{attribute 'linkalways'} 
{attribute 'no_explicit_call' := 'This FB is a CLASS and must be accessed using methods or properties'}
{attribute 'enable_dynamic_creation'}
FUNCTION_BLOCK _DINT EXTENDS NumericDatatypeBase
VAR
	localData : DINT;
	activeData : REFERENCE TO DINT REF= localData;
END_VAR

PROPERTY PUBLIC Address : PVOID
GET
Address := ADR(activeData);
END_GET
END_PROPERTY

METHOD PUBLIC ClearReference
VAR_INPUT
END_VAR
activeData REF= localData;
END_METHOD

METHOD PUBLIC Clone : I_Datatype
VAR
    pClone : POINTER TO _DINT;
END_VAR
pClone := __NEW(_DINT(InitialValue := Value));
Clone := pClone^;
END_METHOD

METHOD FB_init : BOOL
VAR_INPUT
	bInitRetains : BOOL; // if TRUE, the retain variables are initialized (warm start / cold start)
	bInCopyCode : BOOL;  // if TRUE, the instance afterwards gets moved into the copy code (online change)
	InitialValue : DINT;
END_VAR
localData := InitialValue;
END_METHOD

PROPERTY PUBLIC IsFloat : BOOL
GET
IsFloat := FALSE;
END_GET
END_PROPERTY

PROPERTY PUBLIC IsSigned : BOOL
GET
IsSigned := TRUE;
END_GET
END_PROPERTY

METHOD PUBLIC MakeReferenceTo
VAR_INPUT
	ReferenceTarget : REFERENCE TO DINT;
END_VAR
activeData REF= ReferenceTarget;
END_METHOD

PROPERTY PUBLIC MaxValue : DINT
GET
MaxValue := DatatypeLimits.DINT_MAX_VALUE;
END_GET
END_PROPERTY

PROPERTY PUBLIC MinValue : DINT
GET
MinValue := DatatypeLimits.DINT_MIN_VALUE;
END_GET
END_PROPERTY

METHOD PROTECTED SerializeMaxValue
VAR_INPUT
	Serializer : I_Serializer;
END_VAR
Serializer.AddDint(MaxValue);
END_METHOD

METHOD PROTECTED SerializeMinValue
VAR_INPUT
	Serializer : I_Serializer;
END_VAR
Serializer.AddDint(MinValue);
END_METHOD

METHOD PUBLIC SerializeWith
VAR_INPUT
	Serializer : I_Serializer;
END_VAR
Serializer.AddDint(activeData);
END_METHOD

PROPERTY PUBLIC Size : UDINT
GET
Size := SIZEOF(activeData);
END_GET
END_PROPERTY

METHOD TryDeserializeFrom : BOOL
VAR_INPUT
	Deserializer : I_Deserializer;
	Feedback : I_DeserializerFeedback;
END_VAR
TryDeserializeFrom := Deserializer.TryGetDint(activeData, Feedback);
END_METHOD

METHOD TryMakeReferenceTo : BOOL
VAR_INPUT
	Target : I_Datatype;
END_VAR
VAR
	pTargetData : POINTER TO DINT;
END_VAR
IF NOT (Target.TypeName = TypeName) THEN
	RETURN;
END_IF

pTargetData := Target.Address;
activeData REF= pTargetData^;
TryMakeReferenceTo := TRUE;
END_METHOD

PROPERTY PUBLIC TypeName : T_MAXSTRING
GET
TypeName := 'DINT';
END_GET
END_PROPERTY

PROPERTY PUBLIC Value : DINT
GET
Value := activeData;
END_GET
SET
activeData := Value;
END_SET
END_PROPERTY

END_FUNCTION_BLOCK

(* stored: Version 1.1.0.1, ProductVersion 3.1.4024.12
   POU _DINT: Id {380d657c-f4d2-4cbd-a092-86b733404599}, SpecialFunc None
   Folder Constructor: Id {00d2ed6f-b203-492d-9b31-3024b32641ee}
   Folder Protected: Id {ecf4ebc3-4349-436e-a9b8-e0b1697f4bc5}
   Property Address: Id {2facbb97-7ee7-4652-8054-e781816802ce}
   Get Get: Id {d3f8b41a-4e80-431f-afac-1537e78d5597}
   Method ClearReference: Id {d6b2a1f0-8fcf-48f5-9e77-b1f5489c4bb8}
   Method Clone: Id {43148a3d-6fe2-4b50-a82f-2439c5d279dc}
   Method FB_init: Id {9451102f-06b8-4076-aaf6-d3e7b6d2e67e}
   Property IsFloat: Id {a2770302-76c3-47ff-96f0-e135c0343a20}
   Get Get: Id {f6b49c6a-b70f-4218-8a09-0f3d72c9e900}
   Property IsSigned: Id {4c31e323-4195-42f1-ab79-9c1e4675e934}
   Get Get: Id {a0aecc8e-5f09-418e-a31e-8d8c59e41bae}
   Method MakeReferenceTo: Id {9ca0e839-84c3-45f0-8c2c-ab4b76af4678}
   Property MaxValue: Id {a9dddddf-3da4-4484-b5ee-ad4316db854d}
   Get Get: Id {bd9ec948-5b40-4c18-826c-7a50cc60ece5}
   Property MinValue: Id {854646a4-4909-4393-b765-aee98da4c4f8}
   Get Get: Id {9ea1f859-444a-4a05-a354-9bec25d45a7e}
   Method SerializeMaxValue: Id {433b5ad3-825c-4be3-a6ab-a480fa0e62b2}
   Method SerializeMinValue: Id {b2bcce4c-c0d7-4ec2-9247-8d0b2a8cb12c}
   Method SerializeWith: Id {09df2fa5-41ef-43a0-8d6d-ea6375473c4a}
   Property Size: Id {95811da6-1f1f-43a5-9963-c63b490601a0}
   Get Get: Id {6cec5852-9028-434d-983a-7051bfe14f63}
   Method TryDeserializeFrom: Id {ed08c0f2-98c3-43e9-9701-278f8392bf1d}
   Method TryMakeReferenceTo: Id {5d9d49df-cace-4251-bb85-92e58fd5c92d}
   Property TypeName: Id {a7e1e47f-f85a-4c4f-8596-d73ca705520b}
   Get Get: Id {14c870d5-1cc0-434c-80ac-8cef42900a9f}
   Property Value: Id {143cefd9-506d-4f16-b4d7-df36cfcf1da1}
   Get Get: Id {b5deafde-4c2b-43fb-b4a5-5a24a3b98908}
   Set Set: Id {2bc12464-da20-4a99-96e0-d99256d92379} *)
